Staubli VAL3: Custom.dtx

mdesc mNomSpeed
bool bDebug
dio dAlarm = {link=ModbusSrv-0\Modbus-Bit\UsIn_bNull1}
dio dSafety1 = {link=ModbusSrv-0\Modbus-Bit\In2_bNull2}
dio dSafety2 = {link=ModbusSrv-0\Modbus-Bit\UsIn_bNull3}
dio dSaftey3 = {link=ModbusSrv-0\Modbus-Bit\UsIn_bNull3}
dio dSaftey4 = {link=ModbusSrv-0\Modbus-Bit\UsO_bNull5}
dio dSation1
dio dSation2
dio dSation3
dio dSation4
